(* IEC 61131-3 sources: collections/src/Stack, 4 files *)

(* ---- ILifo.st ---- *)
NAMESPACE Simatic.Ax.Collections
    INTERFACE ILifo

        METHOD Push : IListItem
            VAR_INPUT
                item : IListItem;
            END_VAR
        END_METHOD

        METHOD Pop : IListItem
        END_METHOD

        METHOD Top : IListItem
        END_METHOD

        METHOD Count : INT
        END_METHOD

    END_INTERFACE
END_NAMESPACE

(* ---- IStack.st ---- *)
NAMESPACE Siemens.Ax.Collections
    INTERFACE IStack
        METHOD Push : IListItem
            VAR_INPUT
                item : IListItem;
            END_VAR
        END_METHOD
        METHOD Pop : IListItem
        END_METHOD
        METHOD Top : IListItem
        END_METHOD
        METHOD Count : INT END_METHOD
    END_INTERFACE
END_NAMESPACE

(* ---- Lifo.st ---- *)
NAMESPACE Simatic.Ax.Collections
    CLASS Lifo IMPLEMENTS ILifo
        VAR PRIVATE
            _list : LinkedList;
        END_VAR

        METHOD PUBLIC FINAL Push : IListItem
            VAR_INPUT
                item : IListItem;
            END_VAR

            Push := _list.Add(item := item);
        END_METHOD

        METHOD PUBLIC Pop : IListItem
            Pop := _list.Head();
            _list.Remove(_list.Head());
        END_METHOD

        METHOD PUBLIC Count : INT
            Count := _list.Count();
        END_METHOD

        METHOD PUBLIC Top : IListItem
            Top := _list.Head();
        END_METHOD
END_CLASS

END_NAMESPACE

(* ---- Stack.st ---- *)
NAMESPACE Siemens.Ax.Collections
    CLASS Fifo IMPLEMENTS IFifo
        VAR PRIVATE
            _list : LinkedList;
        END_VAR

        METHOD PUBLIC FINAL Write
            VAR_INPUT
                item : IListItem;
            END_VAR

            _list.Add(item := item);
        END_METHOD

        METHOD PUBLIC Read : IListItem
            Read := _list.Tail();
            _list.Remove(_list.Tail());
        END_METHOD

        METHOD PUBLIC Count : INT
            Count := _list.Count();
        END_METHOD
END_CLASS

END_NAMESPACE
